% RSLogix 500 project P8_Pump_Speed_Control.RSS, saved by version 12.00.00.00 %
PROJECT "UNTITLED"    % processor: Bul.1763 MicroLogix 1100 Series B %

PROGRAM FILES
  LAD 2   4 rungs
  LAD 3 "IO"  3 rungs
  LAD 4 "CTRL"  10 rungs

DATA FILES
  O0 OUTPUT  4 elements
  I1 INPUT  6 elements
  S2 STATUS  66 elements
  B3 BINARY  1 elements
  T4 TIMER  1 elements
  C5 COUNTER  1 elements
  R6 CONTROL  1 elements
  N7 INTEGER  6 elements
  F8 FLOAT  2 elements

LADDER 2
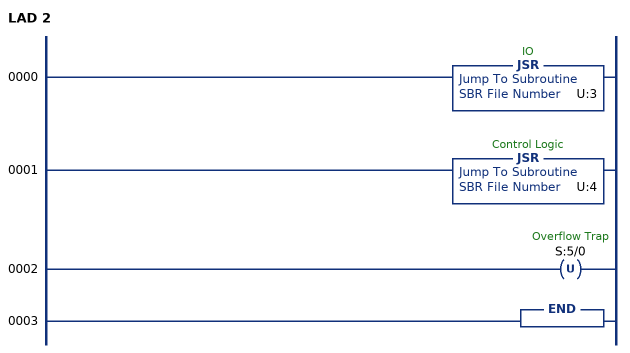
% Rung: 0 %
SOR JSR U:3 EOR
%   U:3  "IO" %
% Rung: 1 %
SOR JSR U:4 EOR
%   U:4  "Control Logic" %
% Rung: 2 %
SOR OTU S:5/0 EOR
%   S:5/0  "Overflow Trap" %
% Rung: 3 %
SOR END EOR

LADDER 3 "IO"
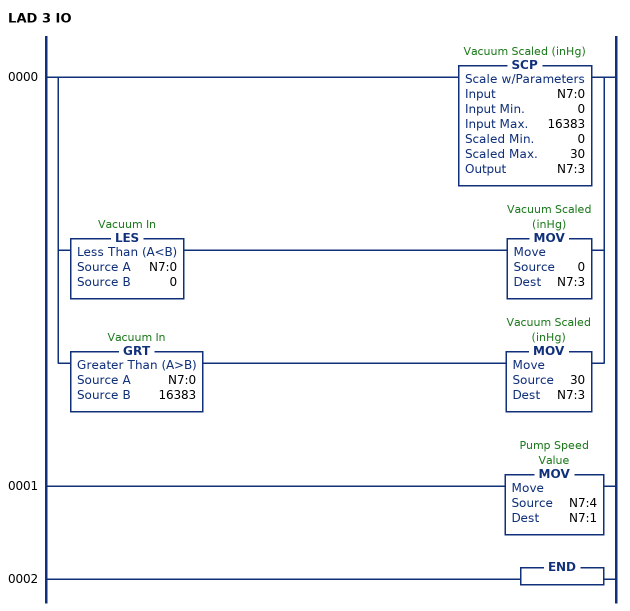
% Rung: 0 %
SOR BST SCP N7:0 0 16383 0 30 N7:3 NXB LES N7:0 0 MOV 0 N7:3 NXB GRT N7:0 16383 MOV 30 N7:3 BND EOR
%   N7:0  "Vacuum In" %
%   N7:3  "Vacuum Scaled (inHg)" %
% Rung: 1 %
SOR MOV N7:4 N7:1 EOR
%   N7:4  "Calculated Pump Speed" %
%   N7:1  "Pump Speed Value" %
% Rung: 2 %
SOR END EOR

LADDER 4 "CTRL"
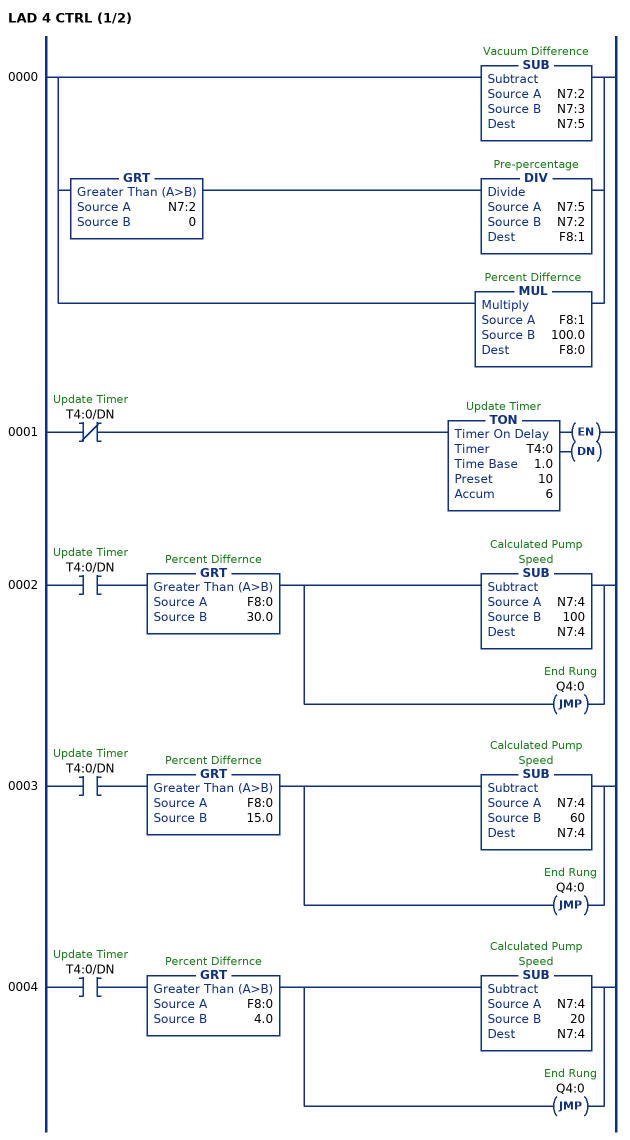
% Rung: 0 %
SOR BST SUB N7:2 N7:3 N7:5 NXB GRT N7:2 0 DIV N7:5 N7:2 F8:1 NXB MUL F8:1 100.0 F8:0 BND EOR
%   N7:3  "Vacuum Scaled (inHg)" %
%   N7:5  "Vacuum Difference" %
%   F8:1  "Pre-percentage" %
%   F8:0  "Percent Differnce" %
% Rung: 1 %
SOR XIO T4:0/DN TON T4:0 1.0 10 6 EOR
%   T4:0  "Update Timer" %
% Rung: 2 %
SOR XIC T4:0/DN GRT F8:0 30.0 BST SUB N7:4 100 N7:4 NXB JMP Q4:0 BND EOR
%   T4:0  "Update Timer" %
%   F8:0  "Percent Differnce" %
%   N7:4  "Calculated Pump Speed" %
%   Q4:0  "End Rung" %
% Rung: 3 %
SOR XIC T4:0/DN GRT F8:0 15.0 BST SUB N7:4 60 N7:4 NXB JMP Q4:0 BND EOR
%   T4:0  "Update Timer" %
%   F8:0  "Percent Differnce" %
%   N7:4  "Calculated Pump Speed" %
%   Q4:0  "End Rung" %
% Rung: 4 %
SOR XIC T4:0/DN GRT F8:0 4.0 BST SUB N7:4 20 N7:4 NXB JMP Q4:0 BND EOR
%   T4:0  "Update Timer" %
%   F8:0  "Percent Differnce" %
%   N7:4  "Calculated Pump Speed" %
%   Q4:0  "End Rung" %

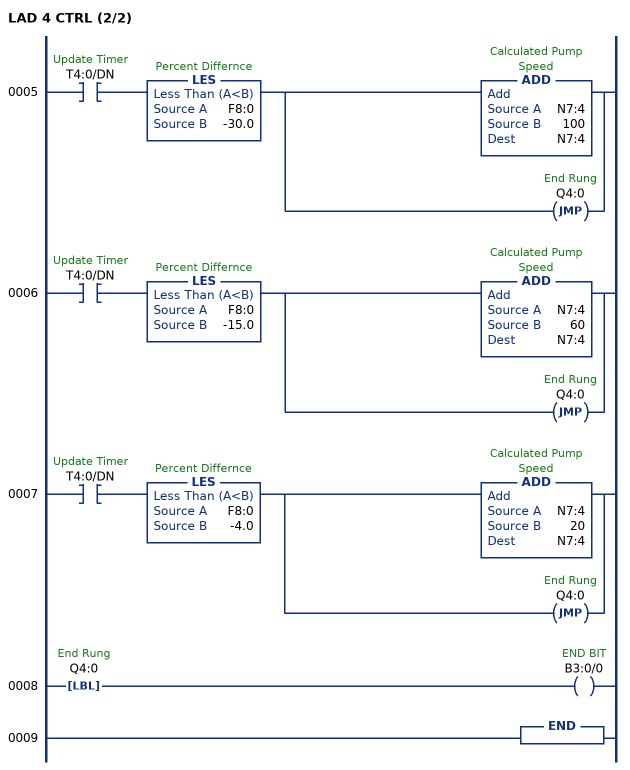
% Rung: 5 %
SOR XIC T4:0/DN LES F8:0 -30.0 BST ADD N7:4 100 N7:4 NXB JMP Q4:0 BND EOR
%   T4:0  "Update Timer" %
%   F8:0  "Percent Differnce" %
%   N7:4  "Calculated Pump Speed" %
%   Q4:0  "End Rung" %
% Rung: 6 %
SOR XIC T4:0/DN LES F8:0 -15.0 BST ADD N7:4 60 N7:4 NXB JMP Q4:0 BND EOR
%   T4:0  "Update Timer" %
%   F8:0  "Percent Differnce" %
%   N7:4  "Calculated Pump Speed" %
%   Q4:0  "End Rung" %
% Rung: 7 %
SOR XIC T4:0/DN LES F8:0 -4.0 BST ADD N7:4 20 N7:4 NXB JMP Q4:0 BND EOR
%   T4:0  "Update Timer" %
%   F8:0  "Percent Differnce" %
%   N7:4  "Calculated Pump Speed" %
%   Q4:0  "End Rung" %
% Rung: 8 %
SOR LBL Q4:0 OTE B3:0/0 EOR
%   Q4:0  "End Rung" %
%   B3:0/0  "END BIT" %
% Rung: 9 %
SOR END EOR

DATA TABLE (non-zero values as saved)
DATA B3
% B3:0 % 0X0001
DATA T4
% .PRE .ACC %
% T4:0 % 10 6
DATA N7
% N7:0 % 4000 200 15 7 200 8
DATA F8
% F8:0 % 53.33334 0.5333334
